// TIA Portal V20 export
// export: Created 2026-04-11T06:02:30.1000377Z, ExportSetting WithDefaults, DisplayName Totally Integrated Automation Portal, DisplayVersion V20, DisplayName TIA Portal Openness, DisplayVersion V20, DisplayName TIA Portal Version Control Interface, DisplayVersion V20, DisplayName STEP 7 Professional, DisplayVersion V20, DisplayName STEP 7 Safety, DisplayVersion V20, DisplayName WinCC Basic/Comfort/Advanced, DisplayVersion V20, DisplayName WinCC Unified, DisplayVersion V20
TYPE "udtError_ModbusTCP"
// stored: IsFailsafeCompliant false
   STRUCT
      bModbusCommError : Bool;   // Modbus transaction attempt timed out
      bModbusMessageError : Bool;   // Address out of range or max lengh exceeded
   END_STRUCT;
END_TYPE
